Staubli VAL3: kill.pgx

public program kill()
begin
  // kill the task create in task PLC and reset the signal
  saveData:bPlcEnable=false
end
